{attribute 'GeneratedUsingTerminal: KL1202'}
{attribute addProperty BoxType "KL1202"}
{attribute addProperty Id "Channel_1AT %Q*Channel_72DF63360Channel_2AT %Q*Channel_72DF63360"}
{attribute addProperty CRC "3968136300"}
{attribute addProperty Size "0"}
TYPE KL1202_EC84F46C :
STRUCT
	{attribute addProperty Name "Channel_1"}
	Channel_1 : Channel_72DF6336;
	{attribute addProperty Name "Channel_2"}
	Channel_2 : Channel_72DF6336;
END_STRUCT
END_TYPE

(* stored: Version 1.2.0.0, ProductVersion 3.1.4024.9
   DUT KL1202_EC84F46C: Id {a1bb6fc5-b5c7-4ce9-9618-9b4f9dd43c98} *)
